FUNCTION_BLOCK FB_MockNciChannelFeedTable EXTENDS FB_ComponentBase IMPLEMENTS I_NciChannel_FeedTable
VAR_INPUT
    MockIsGrouped      : BOOL;
    MockIsReady        : BOOL;
    MockChannelError   : BOOL;
    MockChannelErrorId : UDINT;
    MockIsFeedingDone  : BOOL;
    MockIsChannelDone  : BOOL;
END_VAR
VAR_OUTPUT
    BuildGroupCallCount     : INT;
    StartFeedTableCallCount : INT;
    StopCallCount           : INT;
    UngroupCallCount        : INT;
    ResetCallCount          : INT;
END_VAR

METHOD BuildGroup
BuildGroupCallCount := BuildGroupCallCount + 1;
END_METHOD

PROPERTY ChannelError : BOOL
GET
ChannelError := MockChannelError;
END_GET
END_PROPERTY

PROPERTY ChannelErrorId : UDINT
GET
ChannelErrorId := MockChannelErrorId;
END_GET
END_PROPERTY

PROPERTY IsChannelDone : BOOL
GET
IsChannelDone := MockIsChannelDone;
END_GET
END_PROPERTY

PROPERTY IsFeedingDone : BOOL
GET
IsFeedingDone := MockIsFeedingDone;
END_GET
END_PROPERTY

PROPERTY IsGrouped : BOOL
GET
IsGrouped := MockIsGrouped;
END_GET
END_PROPERTY

PROPERTY IsReady : BOOL
GET
IsReady := MockIsReady;
END_GET
END_PROPERTY

METHOD ResetChannel
ResetCallCount := ResetCallCount + 1;
MockChannelError := FALSE;
MockChannelErrorId := 0;
END_METHOD

METHOD StartFeedTable
VAR_IN_OUT
    stTable : ST_NciFeedGroupTable;
END_VAR
StartFeedTableCallCount := StartFeedTableCallCount + 1;
END_METHOD

METHOD Stop
StopCallCount := StopCallCount + 1;
END_METHOD

METHOD Ungroup
UngroupCallCount := UngroupCallCount + 1;
END_METHOD

END_FUNCTION_BLOCK

(* stored: Version 1.1.0.1, ProductVersion 3.1.4024.15
   POU FB_MockNciChannelFeedTable: Id {d1b2c3d4-e5f6-4789-9999-000000000030}, SpecialFunc None
   Method BuildGroup: Id {a1b2c3d4-e5f6-4789-9999-100000000011}
   Property ChannelError: Id {a1b2c3d4-e5f6-4789-9999-200000000011}
   Get Get: Id {a1b2c3d4-e5f6-4789-9999-200000000012}
   Property ChannelErrorId: Id {a1b2c3d4-e5f6-4789-9999-200000000013}
   Get Get: Id {a1b2c3d4-e5f6-4789-9999-200000000014}
   Property IsChannelDone: Id {a1b2c3d4-e5f6-4789-9999-200000000021}
   Get Get: Id {a1b2c3d4-e5f6-4789-9999-200000000022}
   Property IsFeedingDone: Id {a1b2c3d4-e5f6-4789-9999-200000000019}
   Get Get: Id {a1b2c3d4-e5f6-4789-9999-200000000020}
   Property IsGrouped: Id {a1b2c3d4-e5f6-4789-9999-200000000015}
   Get Get: Id {a1b2c3d4-e5f6-4789-9999-200000000016}
   Property IsReady: Id {a1b2c3d4-e5f6-4789-9999-200000000017}
   Get Get: Id {a1b2c3d4-e5f6-4789-9999-200000000018}
   Method ResetChannel: Id {a1b2c3d4-e5f6-4789-9999-100000000013}
   Method StartFeedTable: Id {a1b2c3d4-e5f6-4789-9999-100000000012}
   Method Stop: Id {a1b2c3d4-e5f6-4789-9999-100000000014}
   Method Ungroup: Id {a1b2c3d4-e5f6-4789-9999-100000000015} *)
